// ============================================
// DB_RecipeProgram1 - Marker Test
// Lines: 53
// CHUNKS: 10 x 100
// Generated by SpinningCam  [2026-09-06 04:29:58]
// ============================================
//
// --- MAKINE AYARLARI ---
// Machine Origin  : X=0.0, Z=0.0
// Axis Direction  : X=NORMAL, Z=NORMAL
// Output Mode     : RADIUS
// G54 Offset      : X=0.0, Z=0.0
// Home            : X=-400.0, Z=-150.0
// Retract         : X=50.0, Z=50.0
//
// --- PARCA / BLANK ---
// Blank Radius    : 0.0 mm
// Blank Z Shift   : 0.0 mm
// Final Thickness : 0.0 mm
// Min Safety Gap  : -999.0 mm
//
// --- MANDREL POZISYON ---
// Mandrel Offset  : X=0.0, Z=0.0
// Mandrel Rot     : Rx=0.0, Ry=0.0, Rz=0.0
//
// --- OPERASYONLAR ---
// Op1: ROUGHING, 3 paso, T0104, R=25.0mm, RPM=600, mm_min=300
// Op2: ROUGHING, 2 paso, T0104, R=25.0mm, RPM=600, mm_min=300
// Op3: ROUGHING, 1 paso, T0104, R=25.0mm, RPM=800, mm_min=200
// Op4: ROUGHING, 3 paso, T0104, R=25.0mm, RPM=0, mm_min=300
// Op5: BENDING, 1 paso, T0104, R=25.0mm, RPM=0, mm_min=300
// ============================================

DATA_BLOCK "DB_RecipeProgram1"
{ S7_Optimized_Access := 'FALSE' }
VERSION : 0.2
UNLINKED
NON_RETAIN
    VAR
        Header : "RecipeHeader";
        Lines1  : Array[0..99] of "RecipeLine";  // global lines 0..99
        Lines2  : Array[0..99] of "RecipeLine";  // global lines 100..199
        Lines3  : Array[0..99] of "RecipeLine";  // global lines 200..299
        Lines4  : Array[0..99] of "RecipeLine";  // global lines 300..399
        Lines5  : Array[0..99] of "RecipeLine";  // global lines 400..499
        Lines6  : Array[0..99] of "RecipeLine";  // global lines 500..599
        Lines7  : Array[0..99] of "RecipeLine";  // global lines 600..699
        Lines8  : Array[0..99] of "RecipeLine";  // global lines 700..799
        Lines9  : Array[0..99] of "RecipeLine";  // global lines 800..899
        Lines10 : Array[0..99] of "RecipeLine";  // global lines 900..999
    END_VAR
BEGIN
    // Header
    Header.sName := 'Marker Test';
    Header.LineCount := 53;
    Header.Valid := TRUE;
    Header.PreScanned := FALSE;
    Header.MinX := 0.000;
    Header.MaxX := 561.676;
    Header.MinZ := 0.000;
    Header.MaxZ := 277.490;

    // --- Tool table (CAM-authored) ---
    Header.ProvidesToolConfig := TRUE;
    Header.ToolCount := 1;
    Header.AutoCalcAngles := TRUE;
    Header.ToolCode_List[1] := 104;
    Header.ToolCode_List[2] := 0;  // unused
    Header.ToolCode_List[3] := 0;  // unused
    Header.ToolCode_List[4] := 0;  // unused
    Header.ToolAngle_List[1] := 0.0;
    Header.ToolAngle_List[2] := 0.0;
    Header.ToolAngle_List[3] := 0.0;
    Header.ToolAngle_List[4] := 0.0;

    // --- Integrity ---
    // Order-sensitive sum over CMD+Param+F of lines 0..LineCount-1.
    // The PLC recomputes it after reassembling the chunks and refuses
    // to run on a mismatch (16#0316). X/Z are excluded on purpose:
    // float32-vs-float64 rounding would eventually cry wolf.
    Header.ProvidesChecksum := TRUE;
    Header.Checksum := 222795;

    // Recipe Lines (53 total)

    // --- Lines1 (global lines 0..52) ---
    Lines1[0].X := 0.000; Lines1[0].Z := 0.000; Lines1[0].F := 5; Lines1[0].CMD := 50; Lines1[0].Param := 1; // OPERATION 1 of 5 [Op1]
    Lines1[1].X := 0.000; Lines1[1].Z := 0.000; Lines1[1].F := 0; Lines1[1].CMD := 10; Lines1[1].Param := 104; // Tool Change T104
    Lines1[2].X := 0.000; Lines1[2].Z := 0.000; Lines1[2].F := 0; Lines1[2].CMD := 20; Lines1[2].Param := 60; // Spindle ON 600 RPM
    Lines1[3].X := 0.000; Lines1[3].Z := 0.000; Lines1[3].F := 3; Lines1[3].CMD := 51; Lines1[3].Param := 1; // PASS 1 of 3 [Op1 P1]
    Lines1[4].X := 480.000; Lines1[4].Z := 110.000; Lines1[4].F := 0; Lines1[4].CMD := 0; Lines1[4].Param := 0; // G0 Rapid [Op1 P1]
    Lines1[5].X := 480.000; Lines1[5].Z := 159.063; Lines1[5].F := 300; Lines1[5].CMD := 1; Lines1[5].Param := 0; // G1 Linear [Op1 P1]
    Lines1[6].X := 480.720; Lines1[6].Z := 160.600; Lines1[6].F := 300; Lines1[6].CMD := 1; Lines1[6].Param := 0; // G1 Linear [Op1 P1]
    Lines1[7].X := 499.877; Lines1[7].Z := 176.216; Lines1[7].F := 300; Lines1[7].CMD := 1; Lines1[7].Param := 0; // G1 Linear [Op1 P1]
    Lines1[8].X := 511.676; Lines1[8].Z := 182.490; Lines1[8].F := 300; Lines1[8].CMD := 1; Lines1[8].Param := 0; // G1 Linear [Op1 P1]
    Lines1[9].X := 561.676; Lines1[9].Z := 232.490; Lines1[9].F := 0; Lines1[9].CMD := 0; Lines1[9].Param := 0; // G0 Rapid [Op1 P1]
    Lines1[10].X := 0.000; Lines1[10].Z := 0.000; Lines1[10].F := 3; Lines1[10].CMD := 51; Lines1[10].Param := 2; // PASS 2 of 3 [Op1 P2]
    Lines1[11].X := 470.000; Lines1[11].Z := 130.000; Lines1[11].F := 0; Lines1[11].CMD := 0; Lines1[11].Param := 0; // G0 Rapid [Op1 P2]
    Lines1[12].X := 470.000; Lines1[12].Z := 179.063; Lines1[12].F := 300; Lines1[12].CMD := 1; Lines1[12].Param := 0; // G1 Linear [Op1 P2]
    Lines1[13].X := 470.720; Lines1[13].Z := 180.600; Lines1[13].F := 300; Lines1[13].CMD := 1; Lines1[13].Param := 0; // G1 Linear [Op1 P2]
    Lines1[14].X := 489.877; Lines1[14].Z := 196.216; Lines1[14].F := 300; Lines1[14].CMD := 1; Lines1[14].Param := 0; // G1 Linear [Op1 P2]
    Lines1[15].X := 501.676; Lines1[15].Z := 202.490; Lines1[15].F := 300; Lines1[15].CMD := 1; Lines1[15].Param := 0; // G1 Linear [Op1 P2]
    Lines1[16].X := 551.676; Lines1[16].Z := 252.490; Lines1[16].F := 0; Lines1[16].CMD := 0; Lines1[16].Param := 0; // G0 Rapid [Op1 P2]
    Lines1[17].X := 0.000; Lines1[17].Z := 0.000; Lines1[17].F := 3; Lines1[17].CMD := 51; Lines1[17].Param := 3; // PASS 3 of 3 [Op1 P3]
    Lines1[18].X := 460.000; Lines1[18].Z := 150.000; Lines1[18].F := 0; Lines1[18].CMD := 0; Lines1[18].Param := 0; // G0 Rapid [Op1 P3]
    Lines1[19].X := 460.000; Lines1[19].Z := 199.063; Lines1[19].F := 300; Lines1[19].CMD := 1; Lines1[19].Param := 0; // G1 Linear [Op1 P3]
    Lines1[20].X := 460.720; Lines1[20].Z := 200.600; Lines1[20].F := 300; Lines1[20].CMD := 1; Lines1[20].Param := 0; // G1 Linear [Op1 P3]
    Lines1[21].X := 479.877; Lines1[21].Z := 216.216; Lines1[21].F := 300; Lines1[21].CMD := 1; Lines1[21].Param := 0; // G1 Linear [Op1 P3]
    Lines1[22].X := 491.676; Lines1[22].Z := 222.490; Lines1[22].F := 300; Lines1[22].CMD := 1; Lines1[22].Param := 0; // G1 Linear [Op1 P3]
    Lines1[23].X := 541.676; Lines1[23].Z := 272.490; Lines1[23].F := 0; Lines1[23].CMD := 0; Lines1[23].Param := 0; // G0 Rapid [Op1 P3]
    Lines1[24].X := 0.000; Lines1[24].Z := 0.000; Lines1[24].F := 5; Lines1[24].CMD := 50; Lines1[24].Param := 2; // OPERATION 2 of 5 [Op2]
    Lines1[25].X := 0.000; Lines1[25].Z := 0.000; Lines1[25].F := 2; Lines1[25].CMD := 51; Lines1[25].Param := 1; // PASS 1 of 2 [Op2 P1]
    Lines1[26].X := 477.500; Lines1[26].Z := 115.000; Lines1[26].F := 0; Lines1[26].CMD := 0; Lines1[26].Param := 0; // G0 Rapid [Op2 P1]
    Lines1[27].X := 477.500; Lines1[27].Z := 164.063; Lines1[27].F := 300; Lines1[27].CMD := 1; Lines1[27].Param := 0; // G1 Linear [Op2 P1]
    Lines1[28].X := 478.220; Lines1[28].Z := 165.600; Lines1[28].F := 300; Lines1[28].CMD := 1; Lines1[28].Param := 0; // G1 Linear [Op2 P1]
    Lines1[29].X := 497.377; Lines1[29].Z := 181.216; Lines1[29].F := 300; Lines1[29].CMD := 1; Lines1[29].Param := 0; // G1 Linear [Op2 P1]
    Lines1[30].X := 509.176; Lines1[30].Z := 187.490; Lines1[30].F := 300; Lines1[30].CMD := 1; Lines1[30].Param := 0; // G1 Linear [Op2 P1]
    Lines1[31].X := 559.176; Lines1[31].Z := 237.490; Lines1[31].F := 0; Lines1[31].CMD := 0; Lines1[31].Param := 0; // G0 Rapid [Op2 P1]
    Lines1[32].X := 0.000; Lines1[32].Z := 0.000; Lines1[32].F := 2; Lines1[32].CMD := 51; Lines1[32].Param := 2; // PASS 2 of 2 [Op2 P2]
    Lines1[33].X := 457.500; Lines1[33].Z := 155.000; Lines1[33].F := 0; Lines1[33].CMD := 0; Lines1[33].Param := 0; // G0 Rapid [Op2 P2]
    Lines1[34].X := 457.500; Lines1[34].Z := 204.063; Lines1[34].F := 300; Lines1[34].CMD := 1; Lines1[34].Param := 0; // G1 Linear [Op2 P2]
    Lines1[35].X := 458.220; Lines1[35].Z := 205.600; Lines1[35].F := 300; Lines1[35].CMD := 1; Lines1[35].Param := 0; // G1 Linear [Op2 P2]
    Lines1[36].X := 477.377; Lines1[36].Z := 221.216; Lines1[36].F := 300; Lines1[36].CMD := 1; Lines1[36].Param := 0; // G1 Linear [Op2 P2]
    Lines1[37].X := 489.176; Lines1[37].Z := 227.490; Lines1[37].F := 300; Lines1[37].CMD := 1; Lines1[37].Param := 0; // G1 Linear [Op2 P2]
    Lines1[38].X := 539.176; Lines1[38].Z := 277.490; Lines1[38].F := 0; Lines1[38].CMD := 0; Lines1[38].Param := 0; // G0 Rapid [Op2 P2]
    Lines1[39].X := 0.000; Lines1[39].Z := 0.000; Lines1[39].F := 5; Lines1[39].CMD := 50; Lines1[39].Param := 3; // OPERATION 3 of 5 [Op3]
    Lines1[40].X := 539.176; Lines1[40].Z := 277.490; Lines1[40].F := 0; Lines1[40].CMD := 20; Lines1[40].Param := 80; // Spindle ON 800 RPM [Op2 P2]
    Lines1[41].X := 0.000; Lines1[41].Z := 0.000; Lines1[41].F := 1; Lines1[41].CMD := 51; Lines1[41].Param := 1; // PASS 1 of 1 [Op3 P1]
    Lines1[42].X := 475.000; Lines1[42].Z := 120.000; Lines1[42].F := 0; Lines1[42].CMD := 0; Lines1[42].Param := 0; // G0 Rapid [Op3 P1]
    Lines1[43].X := 475.000; Lines1[43].Z := 169.063; Lines1[43].F := 200; Lines1[43].CMD := 1; Lines1[43].Param := 0; // G1 Linear [Op3 P1]
    Lines1[44].X := 475.720; Lines1[44].Z := 170.600; Lines1[44].F := 200; Lines1[44].CMD := 1; Lines1[44].Param := 0; // G1 Linear [Op3 P1]
    Lines1[45].X := 494.877; Lines1[45].Z := 186.216; Lines1[45].F := 200; Lines1[45].CMD := 1; Lines1[45].Param := 0; // G1 Linear [Op3 P1]
    Lines1[46].X := 506.676; Lines1[46].Z := 192.490; Lines1[46].F := 200; Lines1[46].CMD := 1; Lines1[46].Param := 0; // G1 Linear [Op3 P1]
    Lines1[47].X := 556.676; Lines1[47].Z := 242.490; Lines1[47].F := 0; Lines1[47].CMD := 0; Lines1[47].Param := 0; // G0 Rapid [Op3 P1]
    Lines1[48].X := 556.676; Lines1[48].Z := 0.000; Lines1[48].F := 0; Lines1[48].CMD := 0; Lines1[48].Param := 0; // G0 Rapid [Op3 P1]
    Lines1[49].X := 0.000; Lines1[49].Z := 0.000; Lines1[49].F := 0; Lines1[49].CMD := 0; Lines1[49].Param := 0; // G0 Rapid [Op3 P1]
    Lines1[50].X := 0.000; Lines1[50].Z := 0.000; Lines1[50].F := 0; Lines1[50].CMD := 21; Lines1[50].Param := 0; // Spindle OFF [Op3 P1]
    Lines1[51].X := 0.000; Lines1[51].Z := 0.000; Lines1[51].F := 0; Lines1[51].CMD := 21; Lines1[51].Param := 0; // Spindle OFF
    Lines1[52].X := 0.000; Lines1[52].Z := 0.000; Lines1[52].F := 0; Lines1[52].CMD := 99; Lines1[52].Param := 0; // Program END
END_DATA_BLOCK